FUNCTION_BLOCK FB_Motion
VAR_INPUT
	
END_VAR
VAR_OUTPUT

END_VAR
VAR
	fbMcPower	: MC_Power;
	fbMcJog		: MC_Jog;
	fbMcReset: MC_Reset;
	fbMcStop: MC_Stop;
	fbMcMoveAbs: MC_MoveAbsolute;
	fbMcGearInPos: MC_GearInPos;
	fbMcMoveModulo: MC_MoveModulo;
	fbMcGearOut: MC_GearOut;
	fbMcReadStatus: MC_ReadStatus;
	fbMcSetPosition: MC_SetPosition;
END_VAR
VAR_IN_OUT
	stAxis	: ST_Axis;
	Axis	: AXIS_REF;
	Slave	: AXIS_REF;
END_VAR

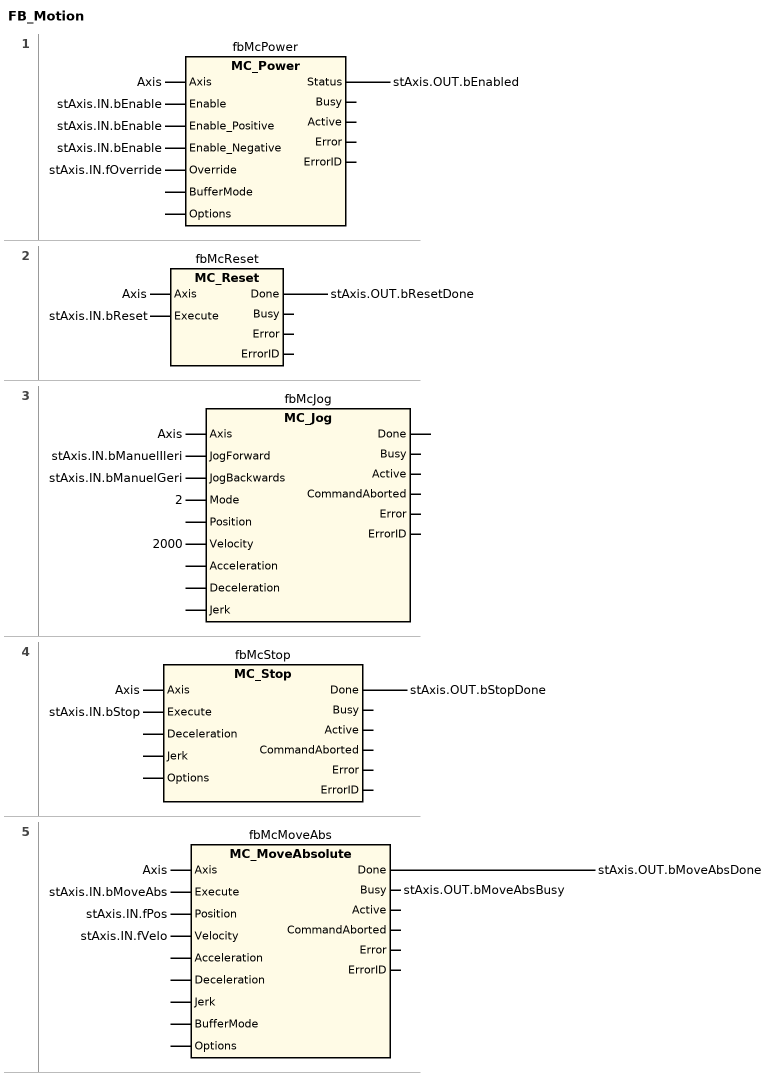
// NETWORK 1
fbMcPower(
    Axis := Axis,
    Enable := stAxis.IN.bEnable,
    Enable_Positive := stAxis.IN.bEnable,
    Enable_Negative := stAxis.IN.bEnable,
    Override := stAxis.IN.fOverride); // MC_Power
stAxis.OUT.bEnabled := fbMcPower.Status;

// NETWORK 2
fbMcReset(Axis := Axis, Execute := stAxis.IN.bReset); // MC_Reset
stAxis.OUT.bResetDone := fbMcReset.Done;

// NETWORK 3
fbMcJog(
    Axis := Axis,
    JogForward := stAxis.IN.bManuelIleri,
    JogBackwards := stAxis.IN.bManuelGeri,
    Mode := 2,
    Velocity := 2000); // MC_Jog

// NETWORK 4
fbMcStop(Axis := Axis, Execute := stAxis.IN.bStop); // MC_Stop
stAxis.OUT.bStopDone := fbMcStop.Done;

// NETWORK 5
fbMcMoveAbs(
    Axis := Axis,
    Execute := stAxis.IN.bMoveAbs,
    Position := stAxis.IN.fPos,
    Velocity := stAxis.IN.fVelo,
    Busy => stAxis.OUT.bMoveAbsBusy); // MC_MoveAbsolute
stAxis.OUT.bMoveAbsDone := fbMcMoveAbs.Done;

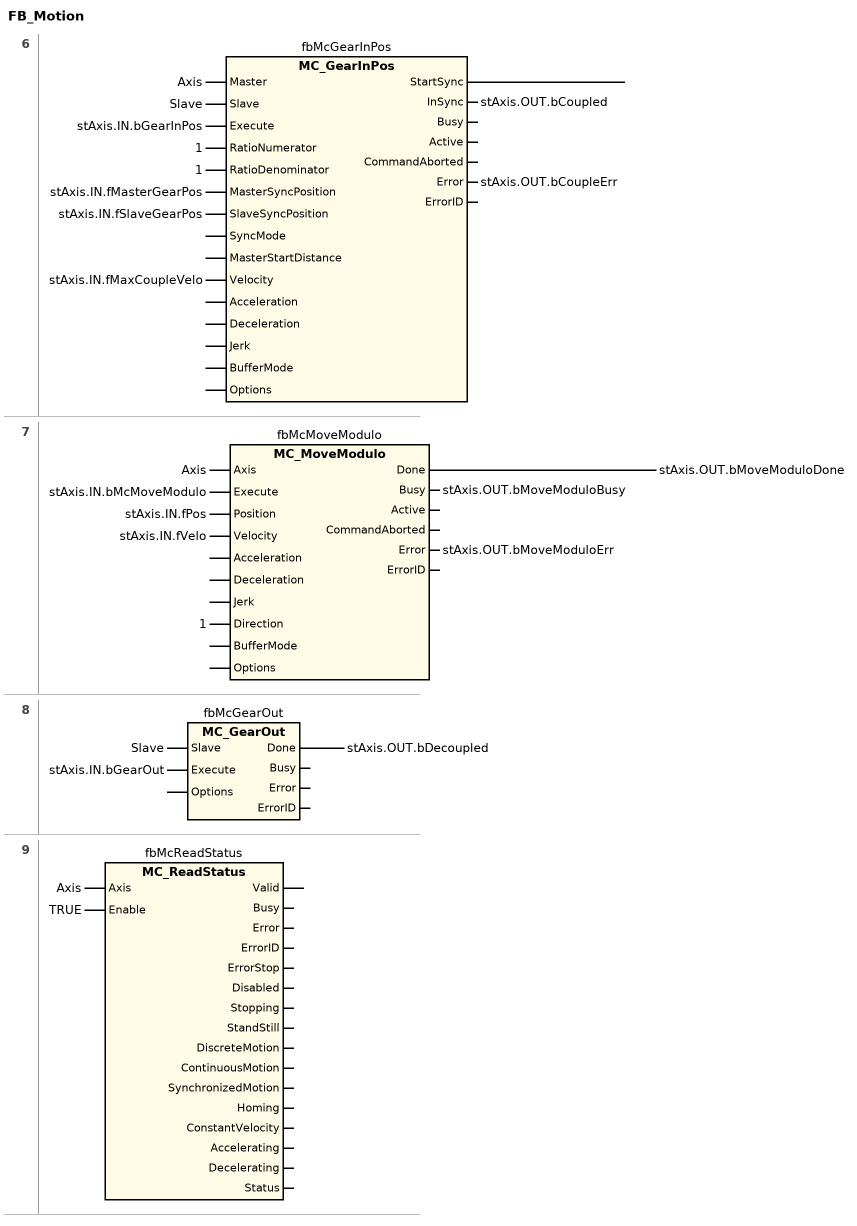
// NETWORK 6
fbMcGearInPos(
    Master := Axis,
    Slave := Slave,
    Execute := stAxis.IN.bGearInPos,
    RatioNumerator := 1,
    RatioDenominator := 1,
    MasterSyncPosition := stAxis.IN.fMasterGearPos,
    SlaveSyncPosition := stAxis.IN.fSlaveGearPos,
    Velocity := stAxis.IN.fMaxCoupleVelo,
    InSync => stAxis.OUT.bCoupled,
    Error => stAxis.OUT.bCoupleErr); // MC_GearInPos

// NETWORK 7
fbMcMoveModulo(
    Axis := Axis,
    Execute := stAxis.IN.bMcMoveModulo,
    Position := stAxis.IN.fPos,
    Velocity := stAxis.IN.fVelo,
    Direction := 1,
    Busy => stAxis.OUT.bMoveModuloBusy,
    Error => stAxis.OUT.bMoveModuloErr); // MC_MoveModulo
stAxis.OUT.bMoveModuloDone := fbMcMoveModulo.Done;

// NETWORK 8
fbMcGearOut(Slave := Slave, Execute := stAxis.IN.bGearOut); // MC_GearOut
stAxis.OUT.bDecoupled := fbMcGearOut.Done;

// NETWORK 9
fbMcReadStatus(Axis := Axis, Enable := TRUE); // MC_ReadStatus

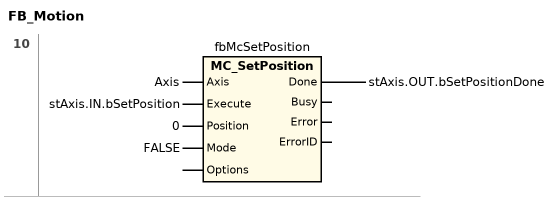
// NETWORK 10
fbMcSetPosition(Axis := Axis, Execute := stAxis.IN.bSetPosition, Position := 0, Mode := FALSE); // MC_SetPosition
stAxis.OUT.bSetPositionDone := fbMcSetPosition.Done;

END_FUNCTION_BLOCK

(* stored: Version 1.1.0.1, ProductVersion 3.1.4022.12
   POU FB_Motion: Id {6f41c403-8015-4d46-9ebe-5eb3fe721611}, SpecialFunc None *)
